FUNCTION fnLogTransfer : BOOL
VAR_INPUT
	logMsgPtr : POINTER TO LogMsg;
END_VAR
VAR
END_VAR


fnLogTransfer := logMsgPtr^.LogTransfer();

END_FUNCTION

(* stored: Version 1.1.0.1, ProductVersion 3.1.4024.3
   POU fnLogTransfer: Id {74a50646-1b73-04e1-357d-a23466a0a7af}, SpecialFunc None *)
